FUNCTION_BLOCK FB_Observer_LREAL EXTENDS FB_AbstractObserver
VAR
    _fVal:              LREAL;
END_VAR

PROPERTY fValue64 : LREAL
GET
fValue64 := THIS^._fVal;
END_GET
END_PROPERTY

{attribute 'hasanytype'}
METHOD Update : I_Observer
VAR_INPUT
    anyVal:         ANY;
END_VAR
Update := THIS^;

IF TO_INT(anyVal.TypeClass) = IBaseLibrary.TypeClass.TYPE_LREAL THEN
    Tc2_System.MEMCPY(destAddr := ADR(THIS^._fVal),
                      srcAddr := anyVal.pValue,
                      n := SIZEOF(THIS^._fVal));
END_IF
END_METHOD

END_FUNCTION_BLOCK

(* stored: Version 1.1.0.1, ProductVersion 3.1.4024.12
   POU FB_Observer_LREAL: Id {18ac8edb-084b-4b9b-99e1-2a47a70cf182}, SpecialFunc None
   Property fValue64: Id {4bfea9c3-3c79-4af7-978b-1f672969750c}
   Get Get: Id {fcc18e89-1db5-47ee-8185-c891c2f049fe}
   Method Update: Id {565f848f-aad1-4f61-afac-661f9ee397df} *)
